FUNCTION_BLOCK FB_RTCVision
VAR
	bFirstCycle			: BOOL := TRUE;	(* First cycle bit *)
	
	(* TCPIP params *)
	sName 				: STRING;		(* TCP/IP device name for other utilities *)
	sHost				: T_IPv4Addr;	(*  *)
	sAmsNetID 			: T_AmsNetID;	(*  *)
	iPort				: UINT;			(*  *)
	tTimeout			: TIME;			(*  *)
	
	(* Internal status *) 
	_bActive			: BOOL;			(* TCP/IP device initialized and ready to work *)
	_bBusy				: BOOL;			(* TCP/IP device is currently proccesing *)
	_bError				: BOOL;			(* Error occured while executing *)
	_iErrorID			: UDINT;		(* Error ID*)
	
	_bJobStarted		: BOOL;
	_bJobStopped		: BOOL;
	_eResult_Station1	: E_VisionResult;
	_eResult_Station2	: E_VisionResult;
	
	eCameraState		: E_RTCCameraState;		(* Current state of camera connection *)
	eCameraInitState	: E_RTCCameraInitState;		(* Current state of camera initialization *)
	eCameraMethodState	: E_RTCCameraMethodState;

	(* TCPIP communicate with Vision System - Service side is role as sever *)
	fbTcpClient 		: FB_TcpClient ;
	
	(* Messages buffers *)
	stSendData							: ST_TcpBufferData;		(*  *)
	stReciveData 						: ST_TcpBufferData;		(*  *)

	(* Temporary messeges *)
	sSendMessage 						: STRING;				(*  *)
	sReciveMessage						: STRING(1000);			(*  *)
	arrBufferMessage					: ARRAY[0..10] OF STRING;
	iMessageIndex	 					: INT;	
	sNewLine							: STRING := '$R$L';
	
	(* Rising edge trigger *)
	rtError								: R_TRIG; 					(* Rising edge trigger for function block error *)
	
	(* Status inormation and number *)
	iLastStatusCode						: INT; 
	sLastStatusCode						: STRING;

	(* Internal variables of methods *)
	eSetJobNumber							: E_VisionJob;
	eGetJobNumber							: E_VisionJob;
	eVisionResult							: E_VisionResult;
	
END_VAR

(* First cycle procedure *)
IF bFirstCycle THEN
	bFirstCycle := FALSE;
	
END_IF

_bActive := eCameraState >= RTC_CAMERA_READY;

(* Report errors that occur *)
rtError(CLK:=_bError);

IF rtError.Q THEN 
	fbMachineLogger.MR_AddLogs(FUN_MergeStrings5(sName, ' : Error occured (error ID: ', UDINT_TO_STRING(_iErrorID), ')', ''));

END_IF

(* Execute TCP/IP FB and timers *)
fbTcpClient();

(* Execute state machine *)
StateMachine();

PROPERTY Active  : REFERENCE TO BOOL
GET
Active REF= _bActive;
END_GET
END_PROPERTY

PROPERTY Busy : REFERENCE TO BOOL
GET
Busy REF= _bBusy;
END_GET
END_PROPERTY

PROPERTY CurrentJob : UINT
GET
END_GET
SET
END_SET
END_PROPERTY

PROPERTY Error : REFERENCE TO BOOL
GET
Error REF= _bError;
END_GET
END_PROPERTY

PROPERTY ErrorID : REFERENCE TO UDINT
GET
ErrorID REF= _iErrorID;
END_GET
END_PROPERTY

METHOD GetInfor : BOOL
VAR_INPUT
END_VAR
END_METHOD

PROPERTY JobStarted : BOOL
GET
END_GET
END_PROPERTY

PROPERTY JobStopped : BOOL
GET
END_GET
END_PROPERTY

METHOD MR_Abort : BOOL
VAR_INPUT
END_VAR
IF eCameraState >= RTC_CAMERA_READY THEN
	_bBusy := TRUE;
	MR_Abort := FALSE;
	eCameraState := RTC_CAMERA_ABORTING;
	fbMachineLogger.MR_AddLogs(CONCAT(sName,' : abort requested'));	
	
ELSIF eCameraState = RTC_CAMERA_UNINITIALIZED THEN
	_bBusy := FALSE;
	MR_Abort := TRUE;
	fbMachineLogger.MR_AddLogs(CONCAT(sName,' : abort done'));	
	
END_IF
END_METHOD

METHOD MR_Clear : BOOL
VAR_INPUT
END_VAR
IF eCameraState = RTC_CAMERA_IDLE THEN
	_bBusy := TRUE;
	MR_Clear := FALSE;
	eCameraState := RTC_CAMERA_CLEAR_DATA;
	fbMachineLogger.MR_AddLogs(CONCAT(sName,' : Clear data requested'));	
	
ELSIF eCameraState = RTC_CAMERA_METHOD_DONE THEN
	_bBusy := FALSE;
	MR_Clear := TRUE;
	fbMachineLogger.MR_AddLogs(CONCAT(sName,' : Clear data done'));	

END_IF
END_METHOD

METHOD MR_FirstCycle : BOOL
VAR_INPUT
	sCameraName 			: STRING;		(*  *)
	sClientHost				: T_IPv4Addr;	(*  *)
	sClientAmsNetID 		: T_AmsNetID;	(*  *)
	iClientPort				: UINT;			(*  *)
	tTimeout				: TIME;			(*  *)
	
END_VAR
(* Set fixture name *)
THIS^.sName := sCameraName;

(* Set fixture server initial parameters *)
THIS^.fbTcpClient.MR_FirstCycle(	sName 		:= CONCAT('TCP/IP client of ',sCameraName),
									sHost		:= sClientHost,
									sAmsNetID	:= sClientAmsNetID,
									iPort 		:= iClientPort,
									tTimeout 	:= tTimeout);
END_METHOD

METHOD MR_GetBatchInfor : BOOL
VAR_INPUT
END_VAR
IF eCameraState = RTC_CAMERA_IDLE THEN	
	_bBusy := TRUE;
	MR_GetBatchInfor := FALSE;
	eCameraState := RTC_CAMERA_GET_BATCH_DATA;
	fbMachineLogger.MR_AddLogs(CONCAT(sName,' : get batch data requested'));
	
ELSIF eCameraState = RTC_CAMERA_METHOD_DONE THEN
	_bBusy := FALSE;
	MR_GetBatchInfor := TRUE;
	fbMachineLogger.MR_AddLogs(CONCAT(sName,' : get batch data done'));

END_IF
END_METHOD

METHOD MR_GetResult : BOOL
VAR_INPUT
END_VAR
IF eCameraState = RTC_CAMERA_IDLE THEN	
	_bBusy := TRUE;
	MR_GetResult := FALSE;
	eCameraState := RTC_CAMERA_GET_RESULT;
	fbMachineLogger.MR_AddLogs(CONCAT(sName,' : get result requested'));
	
ELSIF eCameraState = RTC_CAMERA_METHOD_DONE THEN
	_bBusy := FALSE;
	MR_GetResult := TRUE;
	fbMachineLogger.MR_AddLogs(CONCAT(sName,' : get result done'));

END_IF
END_METHOD

METHOD MR_Init : BOOL
VAR_INPUT
END_VAR
IF eCameraState = RTC_CAMERA_UNINITIALIZED THEN
	_bBusy := TRUE;
	MR_Init := FALSE;
	eCameraState := RTC_CAMERA_INITIALIZING;
	fbMachineLogger.MR_AddLogs(CONCAT(sName,' : initializing requested'));	

ELSIF eCameraState >= RTC_CAMERA_READY THEN
	_bBusy := FALSE;
	MR_Init := TRUE;
	fbMachineLogger.MR_AddLogs(CONCAT(sName,' : initializing done'));
	
END_IF
END_METHOD

METHOD MR_Reset : BOOL
VAR_INPUT
END_VAR
END_METHOD

METHOD MR_SetJob : BOOL
VAR_INPUT
	eSetJobNumber 		: E_VisionJob;
END_VAR
IF eCameraState = RTC_CAMERA_IDLE THEN
	THIS^.eSetJobNumber := eSetJobNumber;
	_bBusy := TRUE;
	MR_SetJob := FALSE;
	eCameraState := RTC_CAMERA_SET_JOB;
	fbMachineLogger.MR_AddLogs(FUN_MergeStrings4(sName,' : setting job ',TO_STRING(eSetJobNumber),' requested'));
	
ELSIF eCameraState = RTC_CAMERA_METHOD_DONE THEN
	_bBusy := FALSE;
	MR_SetJob := TRUE;
	fbMachineLogger.MR_AddLogs(FUN_MergeStrings4(sName,' : setting job ',TO_STRING(eSetJobNumber),' done'));

END_IF
END_METHOD

METHOD MR_Start : BOOL
VAR_INPUT
END_VAR
IF eCameraState = RTC_CAMERA_IDLE THEN
	_bBusy := TRUE;
	MR_Start := FALSE;
	eCameraState := RTC_CAMERA_START;
	fbMachineLogger.MR_AddLogs(CONCAT(sName,' : Start job requested'));	
	
ELSIF eCameraState = RTC_CAMERA_METHOD_DONE THEN
	_bBusy := FALSE;
	MR_Start := TRUE;
	fbMachineLogger.MR_AddLogs(CONCAT(sName,' : Start job done'));	

END_IF
END_METHOD

METHOD MR_Stop : BOOL
VAR_INPUT
END_VAR
IF eCameraState = RTC_CAMERA_IDLE THEN	
	_bBusy := TRUE;
	MR_Stop := FALSE;
	eCameraState := RTC_CAMERA_STOP;
	fbMachineLogger.MR_AddLogs(CONCAT(sName,' : stop job requested'));
	
ELSIF eCameraState = RTC_CAMERA_METHOD_DONE THEN
	_bBusy := FALSE;
	MR_Stop := TRUE;
	fbMachineLogger.MR_AddLogs(CONCAT(sName,' : stop job done'));

END_IF
END_METHOD

METHOD MR_StopCycle : BOOL
VAR_INPUT
END_VAR
IF eCameraState = RTC_CAMERA_IDLE THEN	
	_bBusy := TRUE;
	MR_StopCycle := FALSE;
	eCameraState := RTC_CAMERA_STOP_CYCLE;
	fbMachineLogger.MR_AddLogs(CONCAT(sName,' : stop current cycle requested'));
	
ELSIF eCameraState = RTC_CAMERA_METHOD_DONE THEN
	_bBusy := FALSE;
	MR_StopCycle := TRUE;
	fbMachineLogger.MR_AddLogs(CONCAT(sName,' : stop current cycle done'));

END_IF
END_METHOD

METHOD PROTECTED MS_Aborting
fbTcpClient.MR_Abort();

IF NOT fbTcpClient.Active THEN 
	//IF M_ResetParameters() THEN
		eCameraState := RTC_CAMERA_UNINITIALIZED;
		
	//END_IF	
END_IF
END_METHOD

METHOD PROTECTED MS_GetJob : BOOL
VAR_INPUT
END_VAR
CASE eCameraMethodState OF
	RTC_CAMERA_METHOD_SEND_COMMAND:
		MEMSET(ADR(sSendMessage),0,SIZEOF(sSendMessage));
		sSendMessage := CONCAT('GJ','$R$L');
		FUN_StringToTcpBufferData(ADR(sSendMessage),ADR(stSendData));
		
		IF fbTcpClient.MR_AppendToSendBuffer(stSendData) THEN
			eCameraMethodState := RTC_CAMERA_METHOD_RECEIVE_RESPONSE;

		END_IF
		
	RTC_CAMERA_METHOD_RECEIVE_RESPONSE:
		stReciveData := fbTcpClient.NextRecivedMessage;
		
		IF stReciveData.iLength > 0 THEN
			MEMSET(ADR(sReciveMessage),0,SIZEOF(sReciveMessage));
			FUN_TcpBufferDataToString(ADR(sReciveMessage),ADR(stReciveData));

			IF sReciveMessage = 'GJ1' THEN
				THIS^.eGetJobNumber := CASE_RECEIVER_E25_0100812762;				
			END_IF
			
			eCameraMethodState := RTC_CAMERA_METHOD_SEND_COMMAND;
			eCameraState := RTC_CAMERA_METHOD_DONE;	
		END_IF
		
END_CASE
END_METHOD

METHOD PROTECTED MS_Idle
;
END_METHOD

METHOD PROTECTED MS_Initializing
CASE eCameraInitState OF
	
	RTC_INIT_CONNECTION:
		fbTcpClient.MR_Init();
		
		IF fbTcpClient.Active THEN
			eCameraInitState := RTC_INIT_CLEAR_BUFFER;
			
		ELSIF fbTcpClient.Error THEN
			_bError := TRUE;
			_iErrorID := fbTcpClient.ErrorID;
			
		END_IF
	
	RTC_INIT_CLEAR_BUFFER:
		fbTcpClient.MR_ClearAllBuffers();
		eCameraInitState := RTC_INIT_WAIT_FOR_CONFIRMATION;
		
		IF fbTcpClient.Error THEN
			_bError := TRUE;
			_iErrorID := fbTcpClient.ErrorID;
			
		END_IF

	RTC_INIT_WAIT_FOR_CONFIRMATION:
		stReciveData := fbTcpClient.NextRecivedMessage;

		IF stReciveData.iLength > 0 THEN
			MEMSET(ADR(sReciveMessage),0,SIZEOF(sReciveMessage));
			FUN_TcpBufferDataToString(ADR(sReciveMessage),ADR(stReciveData));
	
			IF sReciveMessage = 'User Logged In' THEN
				eCameraInitState := RTC_INIT_DONE;
			
			END_IF
		ELSIF fbTcpClient.Error THEN
			_bError := TRUE;
			_iErrorID := fbTcpClient.ErrorID;
			
		END_IF
		
	RTC_INIT_DONE:
		eCameraInitState := RTC_INIT_CONNECTION;
		eCameraState := RTC_CAMERA_READY;
END_CASE
END_METHOD

METHOD PROTECTED MS_MethodDone
IF NOT _bBusy THEN
	eCameraState := RTC_CAMERA_IDLE;
	
END_IF
END_METHOD

METHOD PROTECTED MS_Ready
eCameraState := RTC_CAMERA_IDLE;
END_METHOD

METHOD PROTECTED MS_Result
CASE eCameraMethodState OF
	RTC_CAMERA_METHOD_SEND_COMMAND:
		MEMSET(ADR(sSendMessage),0,SIZEOF(sSendMessage));
		sSendMessage := CONCAT('Result','$R$L');
		FUN_StringToTcpBufferData(ADR(sSendMessage),ADR(stSendData));
		
		IF fbTcpClient.MR_AppendToSendBuffer(stSendData) THEN
			eCameraMethodState := RTC_CAMERA_METHOD_RECEIVE_RESPONSE;

		END_IF
		
	RTC_CAMERA_METHOD_RECEIVE_RESPONSE:
		stReciveData := fbTcpClient.NextRecivedMessage;
		
		IF stReciveData.iLength > 0 THEN
			MEMSET(ADR(sReciveMessage),0,SIZEOF(sReciveMessage));
			FUN_TcpBufferDataToString(ADR(sReciveMessage),ADR(stReciveData));
			
			IF sReciveMessage = 'ResultGood' THEN
				eVisionResult := VISION_RESULT_GOOD;
				
			ELSIF sReciveMessage = 'ResultDirt' THEN
				eVisionResult := VISION_RESULT_CONTAMINATION_DIRTY;
				
			ELSIF sReciveMessage = 'ResultDent' THEN
				eVisionResult := VISION_RESULT_SCRATCH_DENT;
				
			ELSIF sReciveMessage = 'ResultReject' THEN
				eVisionResult := VISION_RESULT_REJECT;
				
			ELSE
				eVisionResult := VISION_RESULT_UNKNOWN;
				
			END_IF			
			eCameraMethodState := RTC_CAMERA_METHOD_SEND_COMMAND;
			eCameraState := RTC_CAMERA_METHOD_DONE;	
			
		END_IF		
END_CASE
END_METHOD

METHOD PROTECTED MS_SetJob
CASE eCameraMethodState OF
	RTC_CAMERA_METHOD_SEND_COMMAND:
		MEMSET(ADR(sSendMessage),0,SIZEOF(sSendMessage));
		sSendMessage := FUN_MergeStrings3('SJ', TO_STRING(TO_INT(THIS^.eSetJobNumber)), '$R$L');
		FUN_StringToTcpBufferData(ADR(sSendMessage),ADR(stSendData));
		
		IF fbTcpClient.MR_AppendToSendBuffer(stSendData) THEN
			eCameraMethodState := RTC_CAMERA_METHOD_RECEIVE_RESPONSE;

		END_IF
		
	RTC_CAMERA_METHOD_RECEIVE_RESPONSE:
		stReciveData := fbTcpClient.NextRecivedMessage;
		
		IF stReciveData.iLength > 0 THEN
			MEMSET(ADR(sReciveMessage),0,SIZEOF(sReciveMessage));
			FUN_TcpBufferDataToString(ADR(sReciveMessage),ADR(stReciveData));
			
			IF sReciveMessage = 'SJDone' THEN
				eCameraMethodState := RTC_CAMERA_METHOD_SEND_COMMAND;
				eCameraState := RTC_CAMERA_METHOD_DONE;			
			END_IF	
		END_IF
		
END_CASE
END_METHOD

METHOD PROTECTED MS_Start
CASE eCameraMethodState OF
	
	RTC_CAMERA_METHOD_SEND_COMMAND:
		MEMSET(ADR(sSendMessage),0,SIZEOF(sSendMessage));
		sSendMessage := CONCAT('Start', '$R$L');
		FUN_StringToTcpBufferData(ADR(sSendMessage),ADR(stSendData));
		
		IF fbTcpClient.MR_AppendToSendBuffer(stSendData) THEN
			eCameraMethodState := RTC_CAMERA_METHOD_RECEIVE_RESPONSE;
							
		END_IF
		
	RTC_CAMERA_METHOD_RECEIVE_RESPONSE:
		stReciveData := fbTcpClient.NextRecivedMessage;
		
		IF stReciveData.iLength > 0 THEN
			MEMSET(ADR(sReciveMessage),0,SIZEOF(sReciveMessage));
			FUN_TcpBufferDataToString(ADR(sReciveMessage),ADR(stReciveData));
			
			IF sReciveMessage = 'StartDone' THEN
				eCameraMethodState := RTC_CAMERA_METHOD_SEND_COMMAND;
				eCameraState := RTC_CAMERA_METHOD_DONE;			
			END_IF	
		END_IF

END_CASE
END_METHOD

METHOD PROTECTED MS_Stop : BOOL
VAR_INPUT
END_VAR
CASE eCameraMethodState OF
	RTC_CAMERA_METHOD_SEND_COMMAND:
		MEMSET(ADR(sSendMessage),0,SIZEOF(sSendMessage));
		sSendMessage := CONCAT('Stop','$R$L');
		FUN_StringToTcpBufferData(ADR(sSendMessage),ADR(stSendData));
		
		IF fbTcpClient.MR_AppendToSendBuffer(stSendData) THEN
			eCameraMethodState := RTC_CAMERA_METHOD_RECEIVE_RESPONSE;

		END_IF
		
	RTC_CAMERA_METHOD_RECEIVE_RESPONSE:
		stReciveData := fbTcpClient.NextRecivedMessage;
		
		IF stReciveData.iLength > 0 THEN
			MEMSET(ADR(sReciveMessage),0,SIZEOF(sReciveMessage));
			FUN_TcpBufferDataToString(ADR(sReciveMessage),ADR(stReciveData));
			
			IF sReciveMessage = 'StopDone' THEN
				eCameraMethodState := RTC_CAMERA_METHOD_SEND_COMMAND;
				eCameraState := RTC_CAMERA_METHOD_DONE;			
			END_IF	
		END_IF
		
END_CASE
END_METHOD

METHOD PROTECTED MS_Uninitialized
;
END_METHOD

METHOD PROTECTED StateMachine : BOOL
VAR_INPUT
END_VAR
CASE eCameraState OF
	RTC_CAMERA_UNINITIALIZED:
		MS_Uninitialized();
	
	RTC_CAMERA_INITIALIZING:
		MS_Initializing();
		
	RTC_CAMERA_READY:
		MS_Ready();
		
	RTC_CAMERA_IDLE:
		MS_Idle();
		
	RTC_CAMERA_SET_JOB:
		MS_SetJob();
		

	
	RTC_CAMERA_METHOD_DONE:
		MS_MethodDone();
		
	RTC_CAMERA_ABORTING:
		MS_Aborting();
END_CASE
END_METHOD

END_FUNCTION_BLOCK

(* stored: Version 1.1.0.1, ProductVersion 3.1.4024.9
   POU FB_RTCVision: Id {824bc918-05bb-4b89-ad30-43a88c2cda76}, SpecialFunc None
   Folder FirstCycle: Id {16fc5e85-2ec4-4872-9442-efef1607810a}
   Folder Properties: Id {078b7afe-0419-4579-8830-94f79960bb2a}
   Folder Parameter: Id {c214bb2a-bd41-4761-af3c-cce70871f00e}
   Folder Status: Id {3dc41e3f-331c-4962-95f8-606668cc1fdf}
   Folder Request: Id {319fb7c3-c825-43ac-82a0-79f6b9b9dc0a}
   Folder StateMachine: Id {2cc74067-e497-4607-83ca-346c745bbb97}
   Property Active: Id {42ed5d1a-829f-4523-ac4c-5fcabc20f30d}
   Get Get: Id {097f88e0-cee3-486e-8812-2386b40ea5b7}
   Property Busy: Id {45ab7b77-e6e7-48c3-a403-874d58949966}
   Get Get: Id {390108aa-bca5-4de9-9f42-a22807c4813d}
   Property CurrentJob: Id {74189524-e2d7-459a-92e8-0316755e6bc2}
   Get Get: Id {69cd6aa3-52a4-478b-ac70-94d4fbc69891}
   Set Set: Id {96ac1347-8b2a-447b-af38-6754f1c7b4fa}
   Property Error: Id {c71d3414-cff1-4e8e-94a6-1e18073ee670}
   Get Get: Id {ad32be09-02ae-4b15-92e1-f27feb16fdfd}
   Property ErrorID: Id {97ab9d11-5fda-491b-bb19-c5bd36614004}
   Get Get: Id {b948c467-6970-4704-8d5a-45c64e354d6f}
   Method GetInfor: Id {38f503a2-c742-48e2-b6ec-c4cbcd642d3e}
   Property JobStarted: Id {33a0fdc9-6408-451a-a058-2ea3701df471}
   Get Get: Id {464f0513-e8a2-4b3d-85e9-6317bf3af45d}
   Property JobStopped: Id {f4280290-2964-4f8c-9c89-9540d616c0cf}
   Get Get: Id {3b773e35-d851-4536-b934-0adff9d20c16}
   Method MR_Abort: Id {756fcd1d-1dac-4277-bb51-d63dc5f41d68}
   Method MR_Clear: Id {31582236-d8d2-4ad3-8afe-e3b6d1b21282}
   Method MR_FirstCycle: Id {54d65007-e43a-4972-8019-db4b847b02a9}
   Method MR_GetBatchInfor: Id {80ddcbcc-3107-4c4b-8861-41140dd4600a}
   Method MR_GetResult: Id {5afdba8b-45f6-400a-9f2a-e8c4dc0ba711}
   Method MR_Init: Id {9fceac19-94cd-4f04-9c9a-428be348b03a}
   Method MR_Reset: Id {f4016d5a-9add-4c84-b034-f8e3b2e2805e}
   Method MR_SetJob: Id {598cecc9-3275-436b-b809-88e0586a024b}
   Method MR_Start: Id {ccdbd273-ad10-4ebd-8362-d8c3e662dbbb}
   Method MR_Stop: Id {f9f0a970-f2bc-4617-9d70-3e73490cd0e2}
   Method MR_StopCycle: Id {43756855-bd03-4149-a867-c259d302f9ab}
   Method MS_Aborting: Id {59469cf5-4157-4f56-b242-1c54ec3d324c}
   Method MS_GetJob: Id {a226574a-dde1-45ac-bfcf-5397f359d818}
   Method MS_Idle: Id {0c440fce-6c74-4b20-bf9a-bc86ad90316d}
   Method MS_Initializing: Id {dce27ce5-b4f2-4bf2-9271-0a2d9590e4a1}
   Method MS_MethodDone: Id {dcda2786-3bd7-4c5b-810e-0537da8ca99e}
   Method MS_Ready: Id {9c2ec2f5-59b4-45d8-bc78-07f3279d6028}
   Method MS_Result: Id {0ccc8a23-eb82-45a8-98bb-c4bd66306856}
   Method MS_SetJob: Id {793e5646-f5bf-40cd-97ab-1c4351c0524d}
   Method MS_Start: Id {854e7313-fb57-42f6-a0ef-9867cdb5ee90}
   Method MS_Stop: Id {1455e1a5-79d3-4393-b7b9-a17034762cfb}
   Method MS_Uninitialized: Id {975b444d-e182-4e87-a6d9-2dd2a4cec155}
   Method StateMachine: Id {3c022ea4-89d2-4322-b743-ab8cc1df030e} *)
